// SIMATIC S7-200 project (STEP 7-Micro/WIN), CPU 221 REL 01.10

ORGANIZATION_BLOCK MAIN:OB1
TITLE=
BEGIN
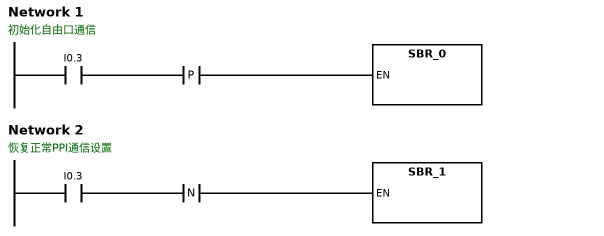
Network 1
// 初始化自由口通信
LD     I0.3
EU
CALL   SBR_0:SBR0
Network 2
// 恢复正常PPI通信设置
LD     I0.3
ED
CALL   SBR_1:SBR1
END_ORGANIZATION_BLOCK

SUBROUTINE_BLOCK SBR_0:SBR0
TITLE=
BEGIN
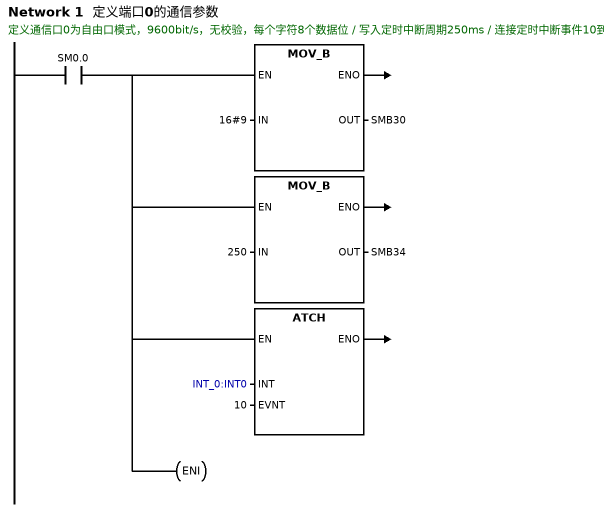
Network 1 // 定义端口0的通信参数
// 定义通信口0为自由口模式，9600bit/s，无校验，每个字符8个数据位
// 写入定时中断周期250ms
// 连接定时中断事件10到中断服务程序INT_0
// 开中断
LD     SM0.0
MOVB   16#9, SMB30
MOVB   250, SMB34
ATCH   INT_0:INT0, 10
ENI
END_SUBROUTINE_BLOCK

SUBROUTINE_BLOCK SBR_1:SBR1
TITLE=
BEGIN
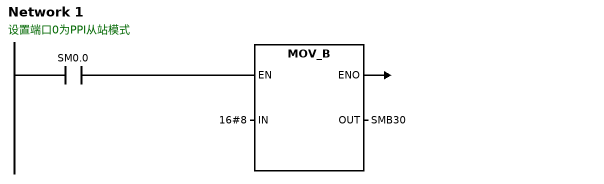
Network 1
// 设置端口0为PPI从站模式
LD     SM0.0
MOVB   16#8, SMB30
END_SUBROUTINE_BLOCK

INTERRUPT_BLOCK INT_0:INT0
TITLE=
BEGIN
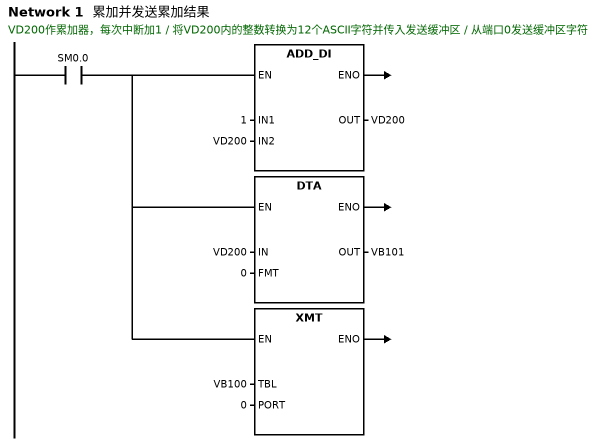
Network 1 // 累加并发送累加结果
// VD200作累加器，每次中断加1
// 将VD200内的整数转换为12个ASCII字符并传入发送缓冲区
// 从端口0发送缓冲区字符
LD     SM0.0
+D     1, VD200
DTA    VD200, VB101, 0
XMT    VB100, 0
END_INTERRUPT_BLOCK

DATA_BLOCK_TAB USER1
BEGIN
//数据块注释
//按F1健获取帮助和示范数据页
VB100    14                  //发送字节数
VD200    0                   //累加器清零
VB113    16#D                //发送数据的结束字符
VB114    16#A                //"回车"的16进制码
END_DATA_BLOCK_TAB
